(* PLC project SafeLOGIC, BrAutomation SafeDESIGNER  5.24.1.0 *)
(* stored: companyURL http://www.br-automation.com, creationDateTime Wed Jan 14 16:08:31 2026 *)

PROGRAM Main

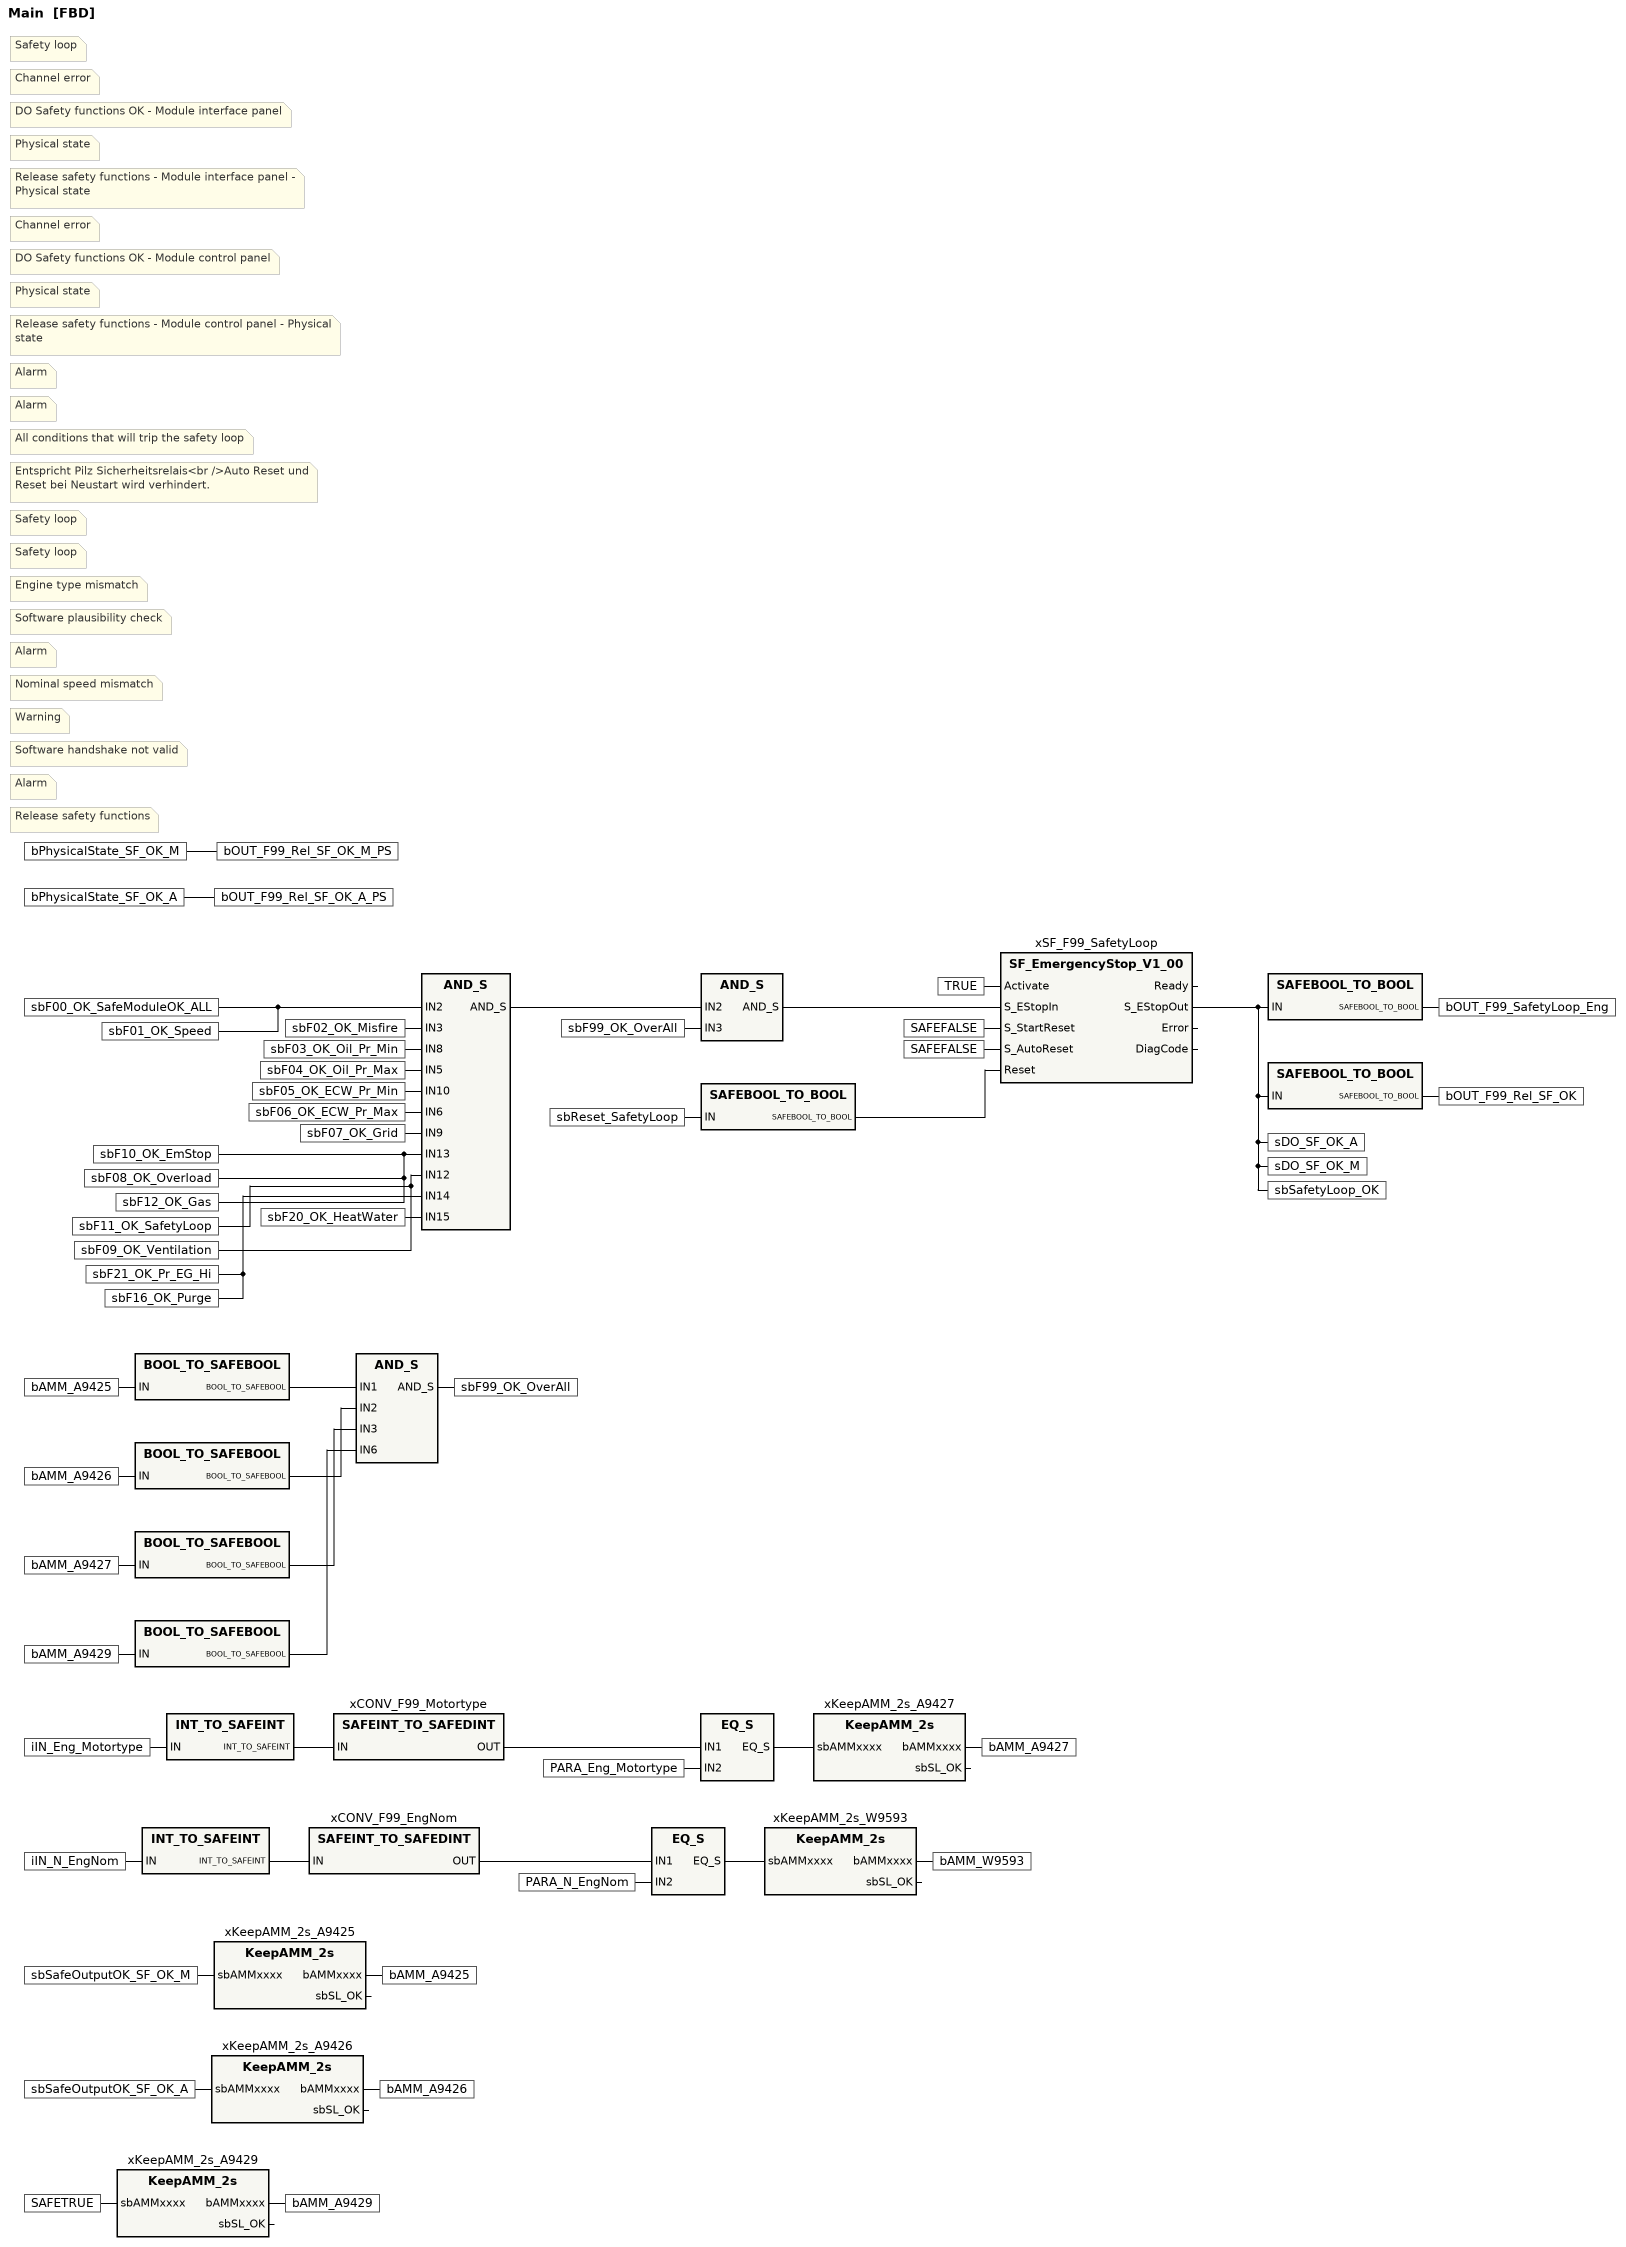
(* FBD diagram, written out as Structured Text *)
(* Safety loop *)
(* DO Safety functions OK - Module interface panel *)
(* Channel error *)
(* Alarm *)
xKeepAMM_2s_A9425(sbAMMxxxx := sbSafeOutputOK_SF_OK_M);
bAMM_A9425 := xKeepAMM_2s_A9425.bAMMxxxx;
(* Physical state *)
(* Release safety functions - Module interface panel - Physical state *)
bOUT_F99_Rel_SF_OK_M_PS := bPhysicalState_SF_OK_M;
(* DO Safety functions OK - Module control panel *)
(* Channel error *)
(* Alarm *)
xKeepAMM_2s_A9426(sbAMMxxxx := sbSafeOutputOK_SF_OK_A);
bAMM_A9426 := xKeepAMM_2s_A9426.bAMMxxxx;
(* Physical state *)
(* Release safety functions - Module control panel - Physical state *)
bOUT_F99_Rel_SF_OK_A_PS := bPhysicalState_SF_OK_A;
(* Software plausibility check *)
(* Engine type mismatch *)
(* Alarm *)
xCONV_F99_Motortype(IN := INT_TO_SAFEINT(iIN_Eng_Motortype));
xKeepAMM_2s_A9427(sbAMMxxxx := EQ_S(xCONV_F99_Motortype.OUT, PARA_Eng_Motortype));
bAMM_A9427 := xKeepAMM_2s_A9427.bAMMxxxx;
(* Nominal speed mismatch *)
(* Warning *)
xCONV_F99_EngNom(IN := INT_TO_SAFEINT(iIN_N_EngNom));
xKeepAMM_2s_W9593(sbAMMxxxx := EQ_S(xCONV_F99_EngNom.OUT, PARA_N_EngNom));
bAMM_W9593 := xKeepAMM_2s_W9593.bAMMxxxx;
(* Software handshake not valid *)
(* Alarm *)
xKeepAMM_2s_A9429(sbAMMxxxx := SAFETRUE);
bAMM_A9429 := xKeepAMM_2s_A9429.bAMMxxxx;
(* Safety loop *)
(* Safety loop *)
sbF99_OK_OverAll := AND_S(BOOL_TO_SAFEBOOL(bAMM_A9425), BOOL_TO_SAFEBOOL(bAMM_A9426), BOOL_TO_SAFEBOOL(bAMM_A9427), BOOL_TO_SAFEBOOL(bAMM_A9429));
(* All conditions that will trip the safety loop *)
(* Entspricht Pilz Sicherheitsrelais<br />Auto Reset und Reset bei Neustart wird verhindert. *)
xSF_F99_SafetyLoop(Activate := TRUE, S_EStopIn := AND_S(AND_S(sbF00_OK_SafeModuleOK_ALL, sbF01_OK_Speed, sbF02_OK_Misfire, sbF03_OK_Oil_Pr_Min, sbF04_OK_Oil_Pr_Max, sbF05_OK_ECW_Pr_Min, sbF06_OK_ECW_Pr_Max, sbF07_OK_Grid, sbF08_OK_Overload, sbF09_OK_Ventilation, sbF10_OK_EmStop, sbF11_OK_SafetyLoop, sbF12_OK_Gas, sbF16_OK_Purge, sbF20_OK_HeatWater, sbF21_OK_Pr_EG_Hi), sbF99_OK_OverAll), S_StartReset := SAFEFALSE, S_AutoReset := SAFEFALSE, Reset := SAFEBOOL_TO_BOOL(sbReset_SafetyLoop));
sDO_SF_OK_A := xSF_F99_SafetyLoop.S_EStopOut;
sDO_SF_OK_M := xSF_F99_SafetyLoop.S_EStopOut;
bOUT_F99_SafetyLoop_Eng := SAFEBOOL_TO_BOOL(xSF_F99_SafetyLoop.S_EStopOut);
sbSafetyLoop_OK := xSF_F99_SafetyLoop.S_EStopOut;
(* Release safety functions *)
bOUT_F99_Rel_SF_OK := SAFEBOOL_TO_BOOL(xSF_F99_SafetyLoop.S_EStopOut);
END_PROGRAM
